Staubli VAL3: setByteAt.pgx

public program setByteAt(num x_nByteIndex, num x_nByte, num& x_nBuffer[])
  local string l_sBinWord
  local num l_nLOword
  local num l_nHIword
  local string l_sTempBinByte
begin

  //gestione del segno???

  if x_nByte<0 or x_nByte>255
    x_nBuffer[x_nByteIndex] = 0
  endIf

  x_nBuffer[x_nByteIndex] = x_nByte

end
